PROGRAM prgComEffIO
VAR
	fbCom		: FB_MqttCommunicator_V3;

END_VAR

fbCom(
	bConnect:= TRUE, 
	strAuthKey:=  'BMS99299754422' ,
	sUserName:= 'f2612c04-11b1-4280-957b-bcd7afeefd1d', 					// adopt MQTT Username
	sUserPassword:= '2b86d9a1-0150-4bd8-8a92-9f5c25a019a3', 				// adopt MQTT Password
	eSavePositionCertificate:= eSavePositionOnPLC.ePostionHardDisk, 
	time_HeartBeat_sec := T#15S,
	bConnected=> , 
	bError=> , 
	hrErrorCode=> , 
	eConnectionState=> , 
	eErrorMessage_Out=> );
(* old
	sUserName:= '003d61dd-570a-4e50-89d6-0c2dba2c04ac', 					// adopt MQTT Username
	sUserPassword:= '40dcd341-b962-41d8-a8f4-5db20343d213', 				// adopt MQTT Password
*)

END_PROGRAM

(* stored: Version 1.1.0.1, ProductVersion 3.1.4024.12
   POU prgComEffIO: Id {cbcd318b-bf51-484c-bcaa-d6efcdf43fe3}, SpecialFunc None *)
